Staubli VAL3: Tool.pjx

--- Tool.pjx ---
Parameters version=s7.8.3 stackSize=5000 millimeterUnit=true
Program file=Edit.pgx
Program file=EnterPageKey.pgx
Program file=getTool.pgx
Program file=Main.pgx
Program file=MainKey.pgx
Program file=OnF1.pgx
Program file=OnF2.pgx
Program file=OnF7.pgx
Program file=OnF8.pgx
Program file=Refresh.pgx
Program file=RefreshList.pgx
Program file=setTool.pgx
Program file=start.pgx
Program file=stop.pgx
Data file=Tool.dtx
Library alias=user path=Disk://userPage/USERPAGE.pjx

--- Tool.dtx ---
bool bExit
bool bListRefresh
bool bUserRefresh
mdesc mNomSpeed
num nSelected
num nType = 1
string sItem = "tool1"
string sList[20]
  [0] = "tool1"
  [1] = "tool2"
  [2] = "tool3"
  [3] = "tool4"
  [4] = "tool5"
  [5] = "tool6"
  [6] = "tool7"
  [7] = "tool8"
  [8] = "tool9"
  [9] = "tool10"
  [10] = "tool11"
  [11] = "tool12"
  [12] = "tool13"
  [13] = "tool14"
  [14] = "tool15"
  [15] = "tool16"
  [16] = "tool17"
  [17] = "tool18"
  [18] = "tool19"
  [19] = "tool20"
string sListItemValue[6]
  [0] = "0    "
  [1] = "0    "
  [2] = "100    "
  [3] = "0    "
  [4] = "0    "
  [5] = "0    "
string sParameter[6]
  [0] = "X        :0        "
  [1] = "Y        :0         "
  [2] = "Z        :100      "
  [3] = "Rx       :0         "
  [4] = "Ry       :0         "
  [5] = "Rz       :0         "
string sToolName
public tool tTool{}
  [tool1] = {z=100, fatherId=flange[0], ioLink=valve1}
  [tool10] = {fatherId=flange[0], ioLink=valve1}
  [tool11] = {fatherId=flange[0], ioLink=valve1}
  [tool12] = {fatherId=flange[0], ioLink=valve1}
  [tool13] = {fatherId=flange[0], ioLink=valve1}
  [tool14] = {fatherId=flange[0], ioLink=valve1}
  [tool15] = {fatherId=flange[0], ioLink=valve1}
  [tool16] = {fatherId=flange[0], ioLink=valve1}
  [tool17] = {fatherId=flange[0], ioLink=valve1}
  [tool18] = {fatherId=flange[0], ioLink=valve1}
  [tool19] = {fatherId=flange[0], ioLink=valve1}
  [tool2] = {fatherId=flange[0], ioLink=valve1}
  [tool20] = {fatherId=flange[0], ioLink=valve1}
  [tool3] = {fatherId=flange[0], ioLink=valve1}
  [tool4] = {fatherId=flange[0], ioLink=valve1}
  [tool5] = {fatherId=flange[0], ioLink=valve1}
  [tool6] = {fatherId=flange[0], ioLink=valve1}
  [tool7] = {fatherId=flange[0], ioLink=valve1}
  [tool8] = {fatherId=flange[0], ioLink=valve1}
  [tool9] = {fatherId=flange[0], ioLink=valve1}

--- Edit.pgx ---
program Edit()
  local bool l_bRes
  local num l_i
  local string l_sValue
  local num l_nSelect
  local string l_sItem
  local num l_nKey
  local num l_nRes
begin

  cls()
  resize(sParameter,1,6)
  sParameter[0]="X"
  sParameter[1]="Y"
  sParameter[2]="Z"
  sParameter[3]="Rx"
  sParameter[4]="Ry"
  sParameter[5]="Rz"
  //
  resize(sListItemValue,1,size(sParameter))
  sListItemValue[0]=toString(".3",tTool[sItem].trsf.x)
  sListItemValue[1]=toString(".3",tTool[sItem].trsf.y)
  sListItemValue[2]=toString(".3",tTool[sItem].trsf.z)
  sListItemValue[3]=toString(".3",tTool[sItem].trsf.rx)
  sListItemValue[4]=toString(".3",tTool[sItem].trsf.ry)
  sListItemValue[5]=toString(".3",tTool[sItem].trsf.rz)
  //
  for l_i=0 to size(sParameter)-1
    call user:strlength(sParameter[l_i],user:nBottomX/2)
    l_sValue=sListItemValue[l_i]
    call user:strlength(l_sValue,user:nBottomX/2+1)
    sParameter[l_i]=sParameter[l_i]+":"+l_sValue
  endFor

  bUserRefresh=true
  bListRefresh=true
  //
  do
    if bUserRefresh
      cls()
      call user:clear(0,13)
      call user:typeMenu(8,"确定")
    endIf
    call user:setList(sItem,sParameter,bUserRefresh,bListRefresh,l_nSelect,l_sItem,l_nKey)
    bUserRefresh=false
    bListRefresh=false
    call EnterPageKey(l_nKey,l_nSelect,sParameter[l_nSelect])
    delay(0)
  until l_nKey==255 or l_nKey==278
  bUserRefresh=true
  bListRefresh=true
end

--- EnterPageKey.pgx ---
program EnterPageKey(num& x_nKey (dimensions=1), num& x_nSelect (dimensions=1), string& x_sItem (dimensions=1))
  local bool l_bRes
  local num l_nItem
  local num l_nKey
  local num l_nView
  local string l_sEmpty
  local string l_sItem
  local string l_sStr
  local string l_sValue
  local string l_sYN[2]
  local point lp
begin
  //
  switch x_nSelect
    case 0
      if x_nKey==270
        call user:editNum(x_sItem,sListItemValue[x_nSelect],tTool[sItem].trsf.x,x_nSelect)
      endIf
    break
    case 1
      if x_nKey==270
        call user:editNum(x_sItem,sListItemValue[x_nSelect],tTool[sItem].trsf.y,x_nSelect)
      endIf
    break
    case 2
      if x_nKey==270
        call user:editNum(x_sItem,sListItemValue[x_nSelect],tTool[sItem].trsf.z,x_nSelect)
      endIf
    break
    case 3
      if x_nKey==270
        call user:editNum(x_sItem,sListItemValue[x_nSelect],tTool[sItem].trsf.rx,x_nSelect)
      endIf
    break
    case 4
      if x_nKey==27
        call user:editNum(x_sItem,sListItemValue[x_nSelect],tTool[sItem].trsf.ry,x_nSelect)
      endIf
    break
    case 5
      if x_nKey==270
        call user:editNum(x_sItem,sListItemValue[x_nSelect],tTool[sItem].trsf.rz,x_nSelect)
      endIf
    break
  endSwitch
  if x_nKey==270
    bUserRefresh=true
    bListRefresh=true
  endIf
end

--- getTool.pgx ---
public program getTool(string& x_sTool, tool& x_tTool)
begin
  x_sTool=sToolName
  x_tTool.trsf=tTool[sToolName].trsf
end

--- MainKey.pgx ---
program MainKey(num x_nKey)
  local num l_nKey
begin
  //
  switch x_nKey
    //
    case 271
      call OnF1()
    break
    //编辑
    case 272
      call OnF2()
    break
    //
    case 273
      //call OnF3()
    break
    //
    case 274
      // call OnF4()
    break
    //
    case 275
    break
    //
    case 276
      //call OnF6()
    break
    //save
    case 277
      call OnF7()
    break
    //返回
    case 278
      call OnF8("是否返回")
    break

  endSwitch
end

--- OnF1.pgx ---
program OnF1()
begin
  //
  if nType==1
    call setTool(sItem)
    popUpMsg("选择工具："+sItem)
  endIf

end

--- OnF2.pgx ---
program OnF2()
begin
  call Edit()
end

--- OnF8.pgx ---
program OnF8(string x_sMsg (dimensions=1))
  local num l_i
  local string l_sYesNo[2]
begin
  l_sYesNo[0]="是"
  l_sYesNo[1]="否"
  call user:questionDialog(x_sMsg,l_sYesNo,l_i)
  if l_i==0 or l_i==1
    bExit=true
  endIf
  bUserRefresh=true
end

--- RefreshList.pgx ---
program RefreshList()
  local num l_ni
begin
  //
  if bListRefresh
    resize(sList,1,20)
    for l_ni=0 to 19
      sList[l_ni]="tool"+toString("",l_ni+1)
    endFor
  endIf

end

--- setTool.pgx ---
public program setTool(string x_sTool)
begin
  //
  sToolName=x_sTool
end
